PROGRAM F33_OuterPrinters
VAR
	aSquareWave		 		: ARRAY[1..2] OF  FB_SquareWave;
	aOuterCodeGenerator 		: ARRAY[1..2] OF  FB_CODE_OuterCodeGenerator;
	aSelectCommand	 		: ARRAY[1..2] OF  FB_PRINTER_SelectCommand;

	aLabelPrintCtrl				: ARRAY[1..2] OF  RS;
	aLabelApplyCtrl			: ARRAY[1..2] OF  RS;

	tonLoweratorAtConstSpeed	: TON;
	rsInhibitLabbeller1Apply		: RS	;
	rsInhibitLabbeller2Apply		: RS	;

	sAppendedString				: T_LongSTRING;
	
	fbDebugCNT				: FB_DEBUG_CounterArray;
	aCNTDebug				: ARRAY [1..10] OF UDINT;
	bResetCNT				: BOOL;
	bEnableResendCommand		: BOOL;
	rtEncoder	: R_TRIG;
END_VAR
VAR // added by the converter: edge detectors and wires of the graphical bodies
    _w1, _w2, _w3, _w4, _w5, _w6 : BOOL;
END_VAR

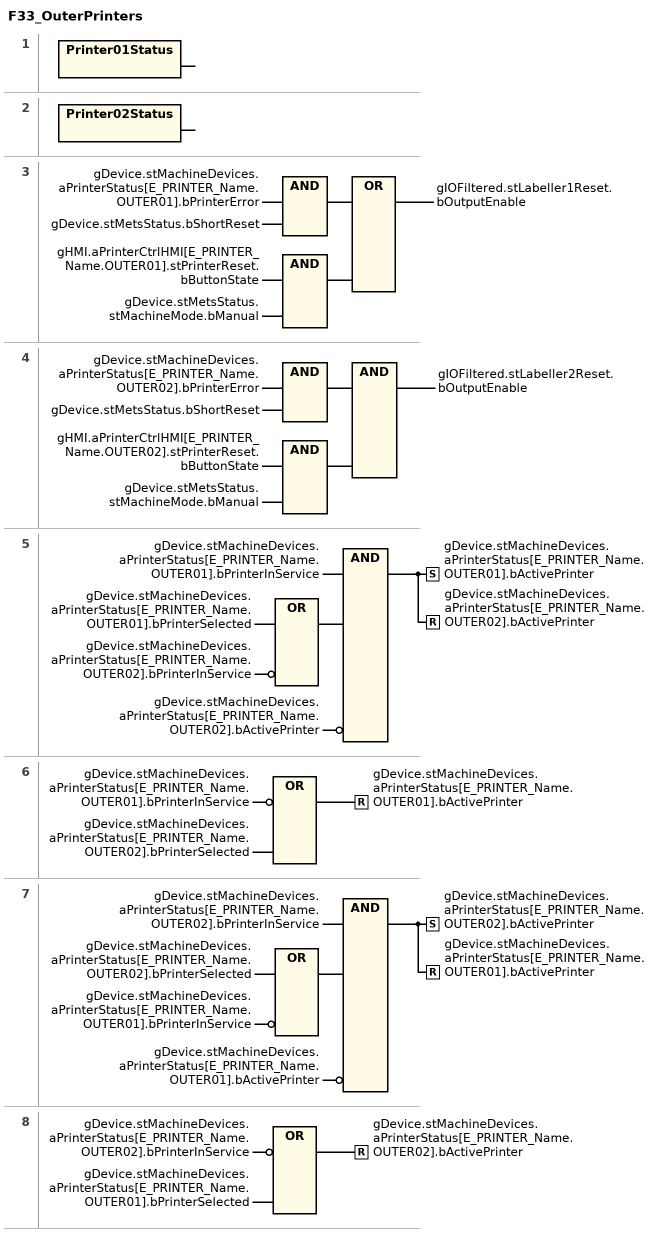
// NETWORK 1
Printer01Status();

// NETWORK 2
Printer02Status();

// NETWORK 3
gIOFiltered.stLabeller1Reset.bOutputEnable := gDevice.stMachineDevices.aPrinterStatus[E_PRINTER_Name.OUTER01].bPrinterError AND gDevice.stMetsStatus.bShortReset OR gHMI.aPrinterCtrlHMI[E_PRINTER_Name.OUTER01].stPrinterReset.bButtonState AND gDevice.stMetsStatus.stMachineMode.bManual;

// NETWORK 4
gIOFiltered.stLabeller2Reset.bOutputEnable := (gDevice.stMachineDevices.aPrinterStatus[E_PRINTER_Name.OUTER02].bPrinterError AND gDevice.stMetsStatus.bShortReset) AND (gHMI.aPrinterCtrlHMI[E_PRINTER_Name.OUTER02].stPrinterReset.bButtonState AND gDevice.stMetsStatus.stMachineMode.bManual);

// NETWORK 5
_w1 := gDevice.stMachineDevices.aPrinterStatus[E_PRINTER_Name.OUTER01].bPrinterInService AND (gDevice.stMachineDevices.aPrinterStatus[E_PRINTER_Name.OUTER01].bPrinterSelected OR NOT gDevice.stMachineDevices.aPrinterStatus[E_PRINTER_Name.OUTER02].bPrinterInService) AND NOT gDevice.stMachineDevices.aPrinterStatus[E_PRINTER_Name.OUTER02].bActivePrinter;
gDevice.stMachineDevices.aPrinterStatus[E_PRINTER_Name.OUTER01].bActivePrinter S= _w1;
gDevice.stMachineDevices.aPrinterStatus[E_PRINTER_Name.OUTER02].bActivePrinter R= _w1;

// NETWORK 6
gDevice.stMachineDevices.aPrinterStatus[E_PRINTER_Name.OUTER01].bActivePrinter R= NOT gDevice.stMachineDevices.aPrinterStatus[E_PRINTER_Name.OUTER01].bPrinterInService OR gDevice.stMachineDevices.aPrinterStatus[E_PRINTER_Name.OUTER02].bPrinterSelected;

// NETWORK 7
_w2 := gDevice.stMachineDevices.aPrinterStatus[E_PRINTER_Name.OUTER02].bPrinterInService AND (gDevice.stMachineDevices.aPrinterStatus[E_PRINTER_Name.OUTER02].bPrinterSelected OR NOT gDevice.stMachineDevices.aPrinterStatus[E_PRINTER_Name.OUTER01].bPrinterInService) AND NOT gDevice.stMachineDevices.aPrinterStatus[E_PRINTER_Name.OUTER01].bActivePrinter;
gDevice.stMachineDevices.aPrinterStatus[E_PRINTER_Name.OUTER02].bActivePrinter S= _w2;
gDevice.stMachineDevices.aPrinterStatus[E_PRINTER_Name.OUTER01].bActivePrinter R= _w2;

// NETWORK 8
gDevice.stMachineDevices.aPrinterStatus[E_PRINTER_Name.OUTER02].bActivePrinter R= NOT gDevice.stMachineDevices.aPrinterStatus[E_PRINTER_Name.OUTER02].bPrinterInService OR gDevice.stMachineDevices.aPrinterStatus[E_PRINTER_Name.OUTER01].bPrinterSelected;

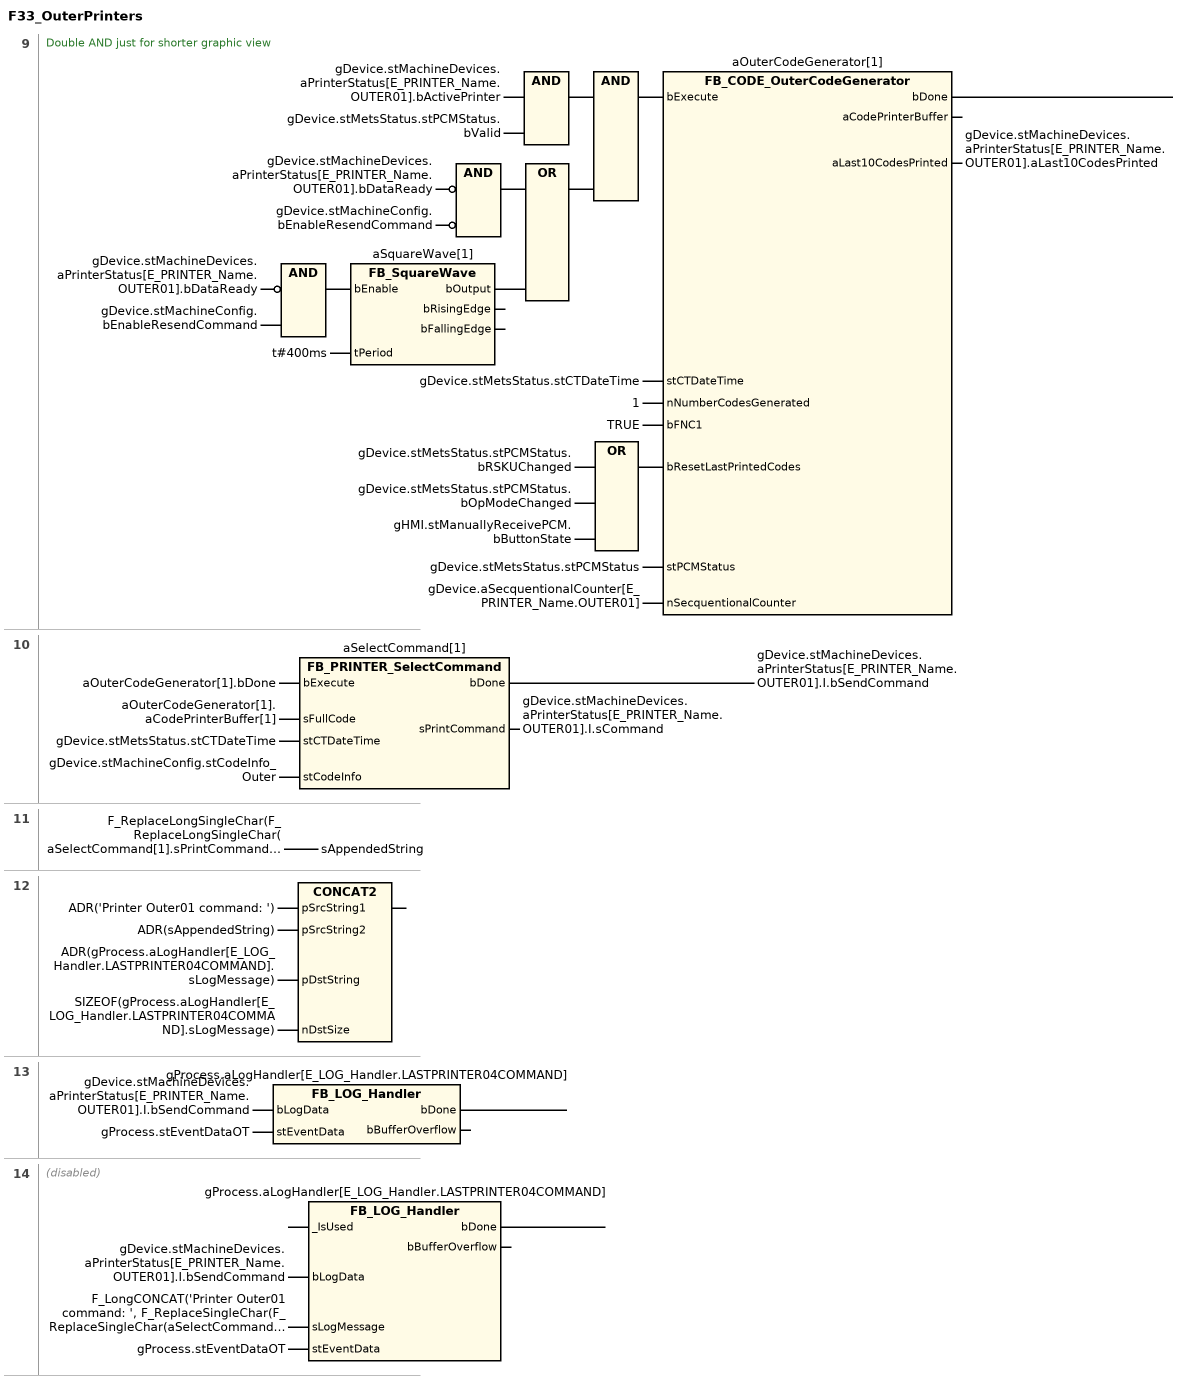
// NETWORK 9
// Double AND just for shorter graphic view
aSquareWave[1](bEnable := NOT gDevice.stMachineDevices.aPrinterStatus[E_PRINTER_Name.OUTER01].bDataReady AND gDevice.stMachineConfig.bEnableResendCommand, tPeriod := t#400ms); // FB_SquareWave
aOuterCodeGenerator[1](
    bExecute := (gDevice.stMachineDevices.aPrinterStatus[E_PRINTER_Name.OUTER01].bActivePrinter AND gDevice.stMetsStatus.stPCMStatus.bValid) AND (NOT gDevice.stMachineDevices.aPrinterStatus[E_PRINTER_Name.OUTER01].bDataReady AND NOT gDevice.stMachineConfig.bEnableResendCommand OR aSquareWave[1].bOutput),
    stCTDateTime := gDevice.stMetsStatus.stCTDateTime,
    nNumberCodesGenerated := 1,
    bFNC1 := TRUE,
    bResetLastPrintedCodes := gDevice.stMetsStatus.stPCMStatus.bRSKUChanged OR gDevice.stMetsStatus.stPCMStatus.bOpModeChanged OR gHMI.stManuallyReceivePCM.bButtonState,
    stPCMStatus := gDevice.stMetsStatus.stPCMStatus,
    nSecquentionalCounter := gDevice.aSecquentionalCounter[E_PRINTER_Name.OUTER01],
    aLast10CodesPrinted => gDevice.stMachineDevices.aPrinterStatus[E_PRINTER_Name.OUTER01].aLast10CodesPrinted); // FB_CODE_OuterCodeGenerator

// NETWORK 10
aSelectCommand[1](
    bExecute := aOuterCodeGenerator[1].bDone,
    sFullCode := aOuterCodeGenerator[1].aCodePrinterBuffer[1],
    stCTDateTime := gDevice.stMetsStatus.stCTDateTime,
    stCodeInfo := gDevice.stMachineConfig.stCodeInfo_Outer,
    sPrintCommand => gDevice.stMachineDevices.aPrinterStatus[E_PRINTER_Name.OUTER01].I.sCommand); // FB_PRINTER_SelectCommand
gDevice.stMachineDevices.aPrinterStatus[E_PRINTER_Name.OUTER01].I.bSendCommand := aSelectCommand[1].bDone;

// NETWORK 11
sAppendedString := F_ReplaceLongSingleChar(F_ReplaceLongSingleChar(aSelectCommand[1].sPrintCommand,'$N','_'),'$R','_');

// NETWORK 12
CONCAT2(pSrcString1 := ADR('Printer Outer01 command: '), pSrcString2 := ADR(sAppendedString), pDstString := ADR(gProcess.aLogHandler[E_LOG_Handler.LASTPRINTER04COMMAND].sLogMessage), nDstSize := SIZEOF(gProcess.aLogHandler[E_LOG_Handler.LASTPRINTER04COMMAND].sLogMessage));

// NETWORK 13
gProcess.aLogHandler[E_LOG_Handler.LASTPRINTER04COMMAND](bLogData := gDevice.stMachineDevices.aPrinterStatus[E_PRINTER_Name.OUTER01].I.bSendCommand, stEventData := gProcess.stEventDataOT); // FB_LOG_Handler

// NETWORK 14 (disabled)
// gProcess.aLogHandler[E_LOG_Handler.LASTPRINTER04COMMAND](
//     bLogData := gDevice.stMachineDevices.aPrinterStatus[E_PRINTER_Name.OUTER01].I.bSendCommand,
//     sLogMessage := F_LongCONCAT('Printer Outer01 command: ', F_ReplaceSingleChar(F_ReplaceSingleChar(aSelectCommand[1].sPrintCommand, '$N', '_' ), '$R', '_')),
//     stEventData := gProcess.stEventDataOT); // FB_LOG_Handler

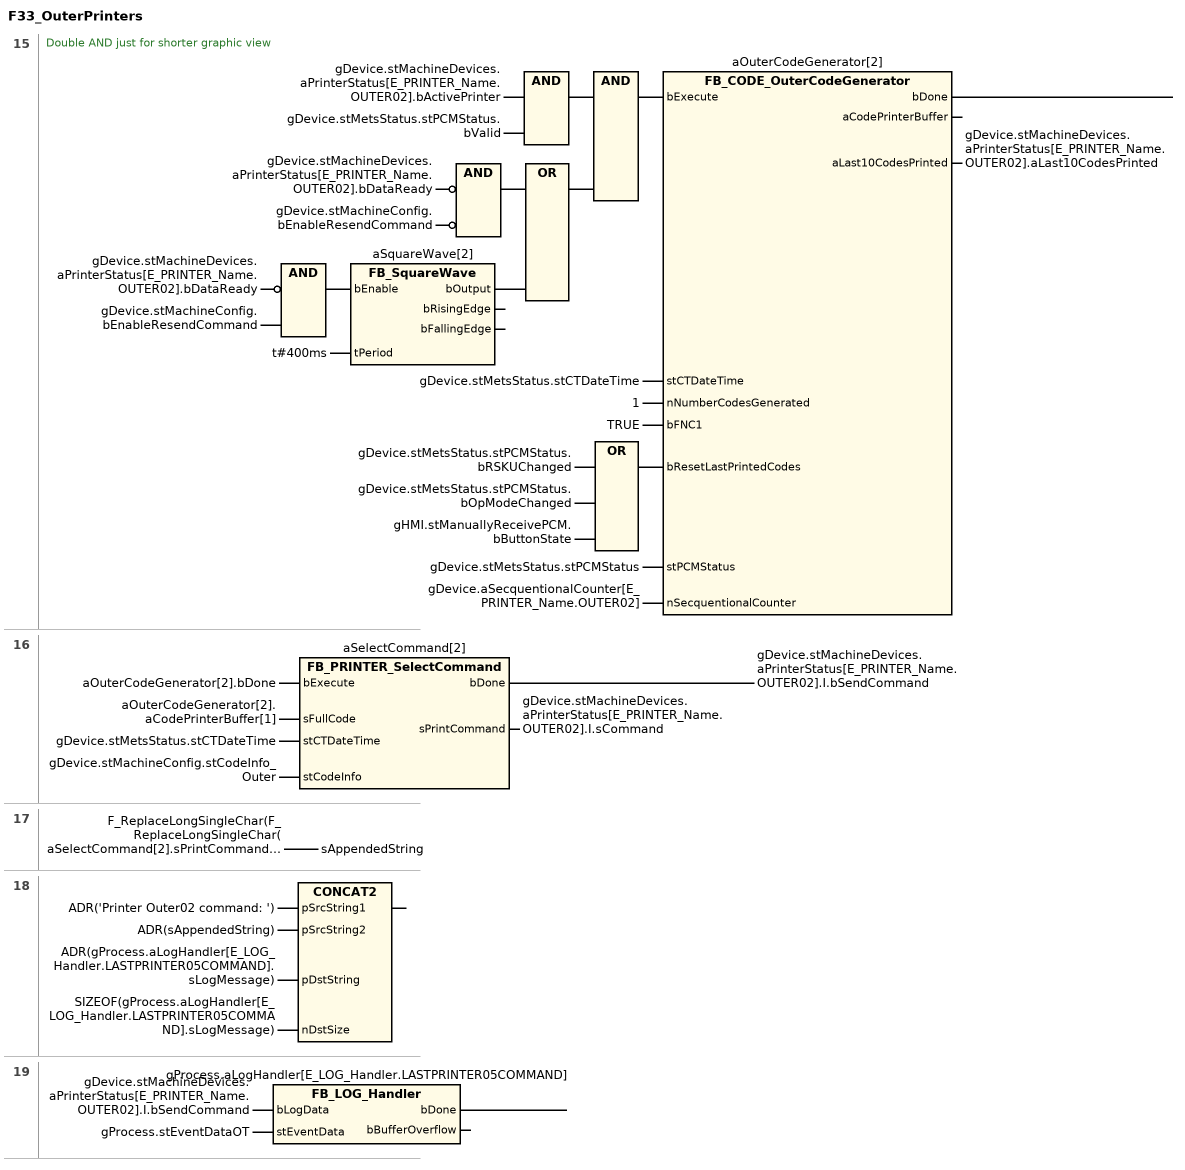
// NETWORK 15
// Double AND just for shorter graphic view
aSquareWave[2](bEnable := NOT gDevice.stMachineDevices.aPrinterStatus[E_PRINTER_Name.OUTER02].bDataReady AND gDevice.stMachineConfig.bEnableResendCommand, tPeriod := t#400ms); // FB_SquareWave
aOuterCodeGenerator[2](
    bExecute := (gDevice.stMachineDevices.aPrinterStatus[E_PRINTER_Name.OUTER02].bActivePrinter AND gDevice.stMetsStatus.stPCMStatus.bValid) AND (NOT gDevice.stMachineDevices.aPrinterStatus[E_PRINTER_Name.OUTER02].bDataReady AND NOT gDevice.stMachineConfig.bEnableResendCommand OR aSquareWave[2].bOutput),
    stCTDateTime := gDevice.stMetsStatus.stCTDateTime,
    nNumberCodesGenerated := 1,
    bFNC1 := TRUE,
    bResetLastPrintedCodes := gDevice.stMetsStatus.stPCMStatus.bRSKUChanged OR gDevice.stMetsStatus.stPCMStatus.bOpModeChanged OR gHMI.stManuallyReceivePCM.bButtonState,
    stPCMStatus := gDevice.stMetsStatus.stPCMStatus,
    nSecquentionalCounter := gDevice.aSecquentionalCounter[E_PRINTER_Name.OUTER02],
    aLast10CodesPrinted => gDevice.stMachineDevices.aPrinterStatus[E_PRINTER_Name.OUTER02].aLast10CodesPrinted); // FB_CODE_OuterCodeGenerator

// NETWORK 16
aSelectCommand[2](
    bExecute := aOuterCodeGenerator[2].bDone,
    sFullCode := aOuterCodeGenerator[2].aCodePrinterBuffer[1],
    stCTDateTime := gDevice.stMetsStatus.stCTDateTime,
    stCodeInfo := gDevice.stMachineConfig.stCodeInfo_Outer,
    sPrintCommand => gDevice.stMachineDevices.aPrinterStatus[E_PRINTER_Name.OUTER02].I.sCommand); // FB_PRINTER_SelectCommand
gDevice.stMachineDevices.aPrinterStatus[E_PRINTER_Name.OUTER02].I.bSendCommand := aSelectCommand[2].bDone;

// NETWORK 17
sAppendedString := F_ReplaceLongSingleChar(F_ReplaceLongSingleChar(aSelectCommand[2].sPrintCommand,'$N','_'),'$R','_');

// NETWORK 18
CONCAT2(pSrcString1 := ADR('Printer Outer02 command: '), pSrcString2 := ADR(sAppendedString), pDstString := ADR(gProcess.aLogHandler[E_LOG_Handler.LASTPRINTER05COMMAND].sLogMessage), nDstSize := SIZEOF(gProcess.aLogHandler[E_LOG_Handler.LASTPRINTER05COMMAND].sLogMessage));

// NETWORK 19
gProcess.aLogHandler[E_LOG_Handler.LASTPRINTER05COMMAND](bLogData := gDevice.stMachineDevices.aPrinterStatus[E_PRINTER_Name.OUTER02].I.bSendCommand, stEventData := gProcess.stEventDataOT); // FB_LOG_Handler

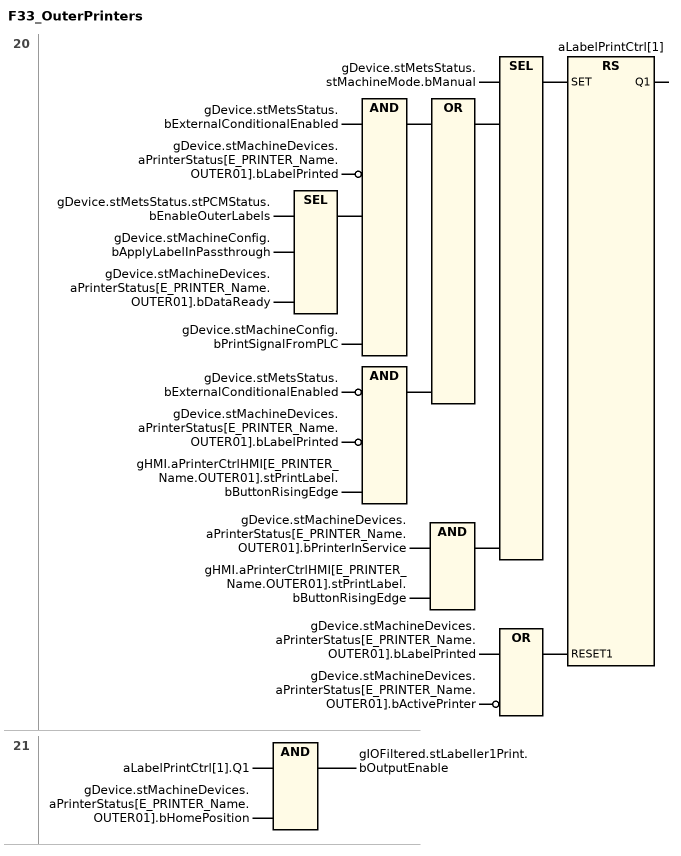
// NETWORK 20
aLabelPrintCtrl[1](SET := SEL(gDevice.stMetsStatus.stMachineMode.bManual, gDevice.stMetsStatus.bExternalConditionalEnabled AND NOT gDevice.stMachineDevices.aPrinterStatus[E_PRINTER_Name.OUTER01].bLabelPrinted AND SEL(gDevice.stMetsStatus.stPCMStatus.bEnableOuterLabels, gDevice.stMachineConfig.bApplyLabelInPassthrough, gDevice.stMachineDevices.aPrinterStatus[E_PRINTER_Name.OUTER01].bDataReady) AND gDevice.stMachineConfig.bPrintSignalFromPLC OR NOT gDevice.stMetsStatus.bExternalConditionalEnabled AND NOT gDevice.stMachineDevices.aPrinterStatus[E_PRINTER_Name.OUTER01].bLabelPrinted AND gHMI.aPrinterCtrlHMI[E_PRINTER_Name.OUTER01].stPrintLabel.bButtonRisingEdge, gDevice.stMachineDevices.aPrinterStatus[E_PRINTER_Name.OUTER01].bPrinterInService AND gHMI.aPrinterCtrlHMI[E_PRINTER_Name.OUTER01].stPrintLabel.bButtonRisingEdge), RESET1 := gDevice.stMachineDevices.aPrinterStatus[E_PRINTER_Name.OUTER01].bLabelPrinted OR NOT gDevice.stMachineDevices.aPrinterStatus[E_PRINTER_Name.OUTER01].bActivePrinter); // RS

// NETWORK 21
gIOFiltered.stLabeller1Print.bOutputEnable := aLabelPrintCtrl[1].Q1 AND gDevice.stMachineDevices.aPrinterStatus[E_PRINTER_Name.OUTER01].bHomePosition;

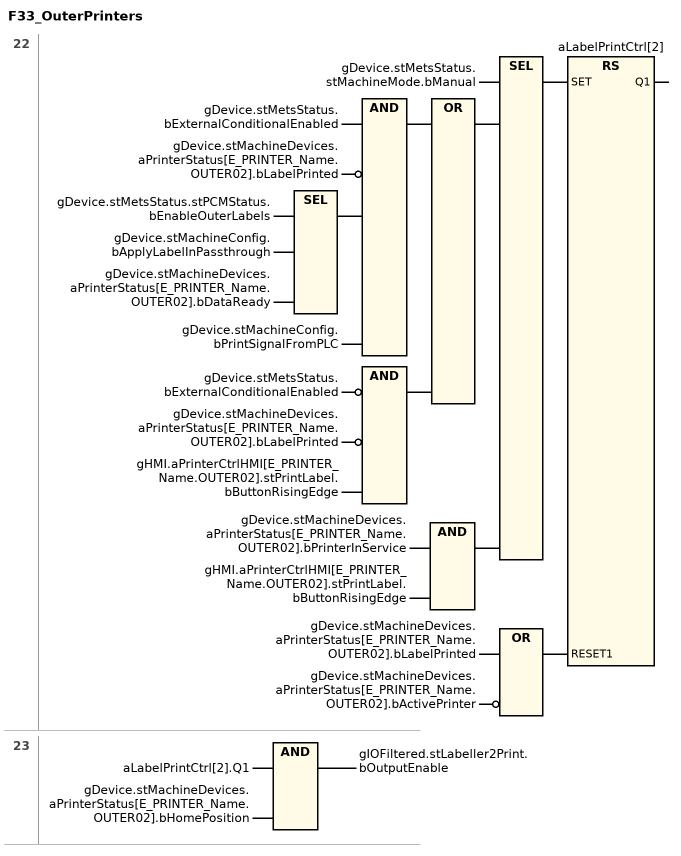
// NETWORK 22
aLabelPrintCtrl[2](SET := SEL(gDevice.stMetsStatus.stMachineMode.bManual, gDevice.stMetsStatus.bExternalConditionalEnabled AND NOT gDevice.stMachineDevices.aPrinterStatus[E_PRINTER_Name.OUTER02].bLabelPrinted AND SEL(gDevice.stMetsStatus.stPCMStatus.bEnableOuterLabels, gDevice.stMachineConfig.bApplyLabelInPassthrough, gDevice.stMachineDevices.aPrinterStatus[E_PRINTER_Name.OUTER02].bDataReady) AND gDevice.stMachineConfig.bPrintSignalFromPLC OR NOT gDevice.stMetsStatus.bExternalConditionalEnabled AND NOT gDevice.stMachineDevices.aPrinterStatus[E_PRINTER_Name.OUTER02].bLabelPrinted AND gHMI.aPrinterCtrlHMI[E_PRINTER_Name.OUTER02].stPrintLabel.bButtonRisingEdge, gDevice.stMachineDevices.aPrinterStatus[E_PRINTER_Name.OUTER02].bPrinterInService AND gHMI.aPrinterCtrlHMI[E_PRINTER_Name.OUTER02].stPrintLabel.bButtonRisingEdge), RESET1 := gDevice.stMachineDevices.aPrinterStatus[E_PRINTER_Name.OUTER02].bLabelPrinted OR NOT gDevice.stMachineDevices.aPrinterStatus[E_PRINTER_Name.OUTER02].bActivePrinter); // RS

// NETWORK 23
gIOFiltered.stLabeller2Print.bOutputEnable := aLabelPrintCtrl[2].Q1 AND gDevice.stMachineDevices.aPrinterStatus[E_PRINTER_Name.OUTER02].bHomePosition;

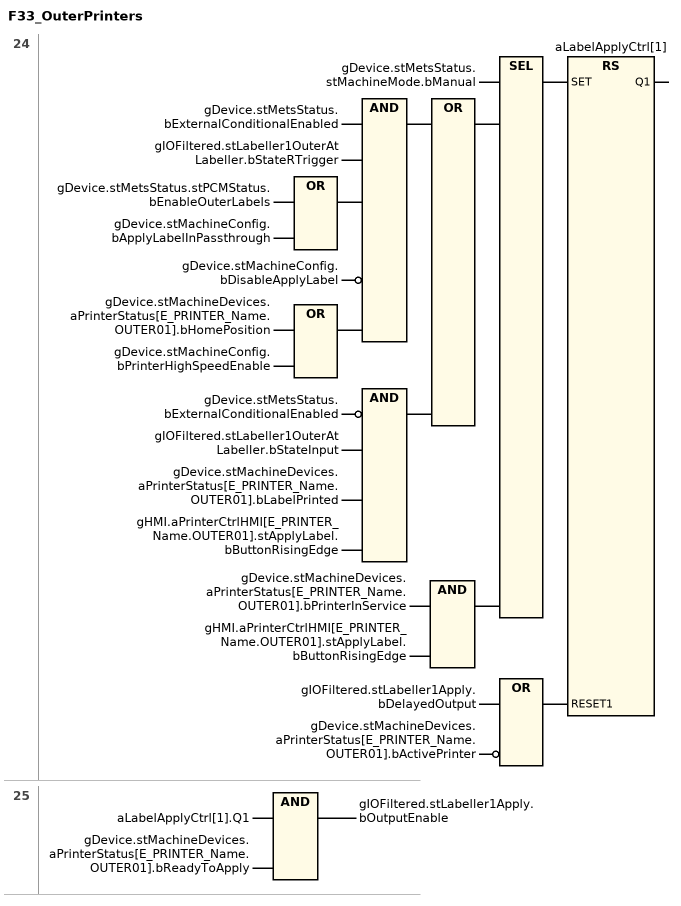
// NETWORK 24
aLabelApplyCtrl[1](SET := SEL(gDevice.stMetsStatus.stMachineMode.bManual, gDevice.stMetsStatus.bExternalConditionalEnabled AND gIOFiltered.stLabeller1OuterAtLabeller.bStateRTrigger AND (gDevice.stMetsStatus.stPCMStatus.bEnableOuterLabels OR gDevice.stMachineConfig.bApplyLabelInPassthrough) AND NOT gDevice.stMachineConfig.bDisableApplyLabel AND (gDevice.stMachineDevices.aPrinterStatus[E_PRINTER_Name.OUTER01].bHomePosition OR gDevice.stMachineConfig.bPrinterHighSpeedEnable) OR NOT gDevice.stMetsStatus.bExternalConditionalEnabled AND gIOFiltered.stLabeller1OuterAtLabeller.bStateInput AND gDevice.stMachineDevices.aPrinterStatus[E_PRINTER_Name.OUTER01].bLabelPrinted AND gHMI.aPrinterCtrlHMI[E_PRINTER_Name.OUTER01].stApplyLabel.bButtonRisingEdge, gDevice.stMachineDevices.aPrinterStatus[E_PRINTER_Name.OUTER01].bPrinterInService AND gHMI.aPrinterCtrlHMI[E_PRINTER_Name.OUTER01].stApplyLabel.bButtonRisingEdge), RESET1 := gIOFiltered.stLabeller1Apply.bDelayedOutput OR NOT gDevice.stMachineDevices.aPrinterStatus[E_PRINTER_Name.OUTER01].bActivePrinter); // RS

// NETWORK 25
gIOFiltered.stLabeller1Apply.bOutputEnable := aLabelApplyCtrl[1].Q1 AND gDevice.stMachineDevices.aPrinterStatus[E_PRINTER_Name.OUTER01].bReadyToApply;

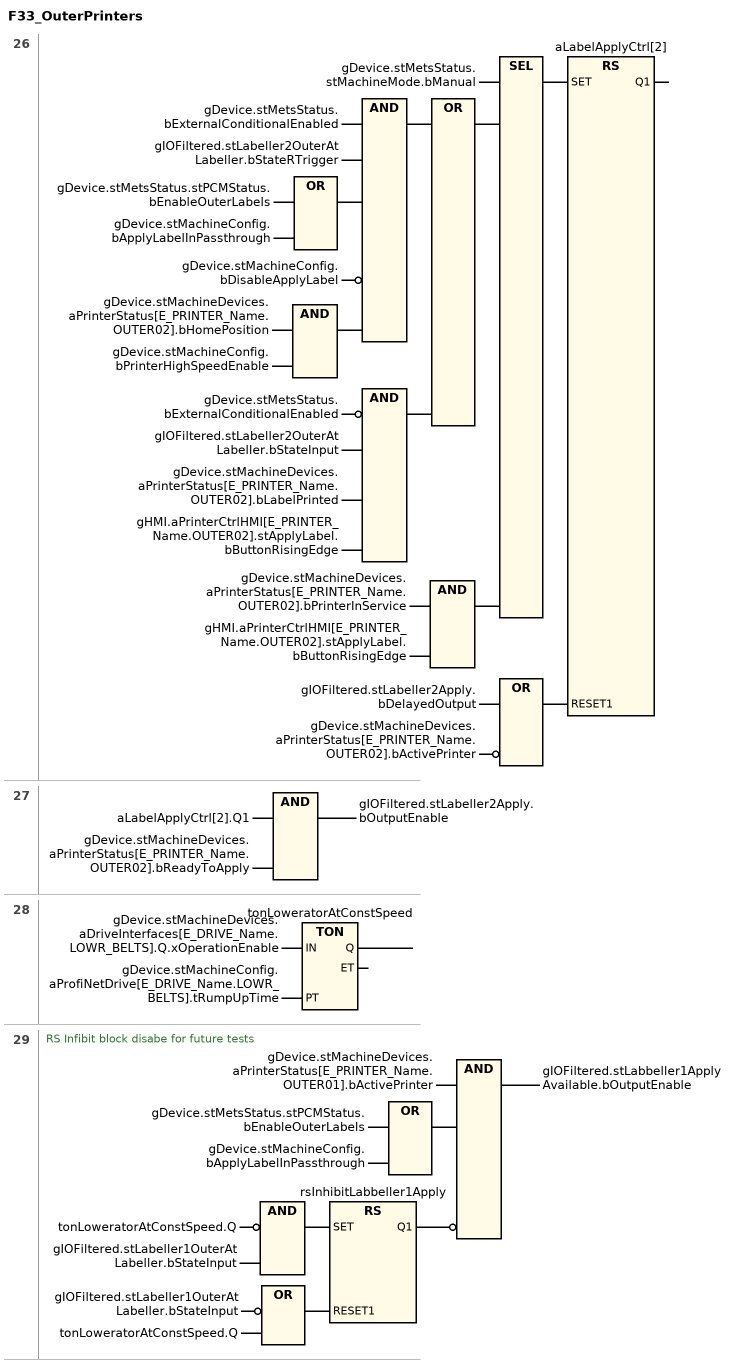
// NETWORK 26
aLabelApplyCtrl[2](SET := SEL(gDevice.stMetsStatus.stMachineMode.bManual, gDevice.stMetsStatus.bExternalConditionalEnabled AND gIOFiltered.stLabeller2OuterAtLabeller.bStateRTrigger AND (gDevice.stMetsStatus.stPCMStatus.bEnableOuterLabels OR gDevice.stMachineConfig.bApplyLabelInPassthrough) AND NOT gDevice.stMachineConfig.bDisableApplyLabel AND (gDevice.stMachineDevices.aPrinterStatus[E_PRINTER_Name.OUTER02].bHomePosition AND gDevice.stMachineConfig.bPrinterHighSpeedEnable) OR NOT gDevice.stMetsStatus.bExternalConditionalEnabled AND gIOFiltered.stLabeller2OuterAtLabeller.bStateInput AND gDevice.stMachineDevices.aPrinterStatus[E_PRINTER_Name.OUTER02].bLabelPrinted AND gHMI.aPrinterCtrlHMI[E_PRINTER_Name.OUTER02].stApplyLabel.bButtonRisingEdge, gDevice.stMachineDevices.aPrinterStatus[E_PRINTER_Name.OUTER02].bPrinterInService AND gHMI.aPrinterCtrlHMI[E_PRINTER_Name.OUTER02].stApplyLabel.bButtonRisingEdge), RESET1 := gIOFiltered.stLabeller2Apply.bDelayedOutput OR NOT gDevice.stMachineDevices.aPrinterStatus[E_PRINTER_Name.OUTER02].bActivePrinter); // RS

// NETWORK 27
gIOFiltered.stLabeller2Apply.bOutputEnable := aLabelApplyCtrl[2].Q1 AND gDevice.stMachineDevices.aPrinterStatus[E_PRINTER_Name.OUTER02].bReadyToApply;

// NETWORK 28
tonLoweratorAtConstSpeed(IN := gDevice.stMachineDevices.aDriveInterfaces[E_DRIVE_Name.LOWR_BELTS].Q.xOperationEnable, PT := gDevice.stMachineConfig.aProfiNetDrive[E_DRIVE_Name.LOWR_BELTS].tRumpUpTime); // TON

// NETWORK 29
// RS Infibit block disabe for future tests
rsInhibitLabbeller1Apply(SET := NOT tonLoweratorAtConstSpeed.Q AND gIOFiltered.stLabeller1OuterAtLabeller.bStateInput, RESET1 := NOT gIOFiltered.stLabeller1OuterAtLabeller.bStateInput OR tonLoweratorAtConstSpeed.Q); // RS
gIOFiltered.stLabbeller1ApplyAvailable.bOutputEnable := gDevice.stMachineDevices.aPrinterStatus[E_PRINTER_Name.OUTER01].bActivePrinter AND (gDevice.stMetsStatus.stPCMStatus.bEnableOuterLabels OR gDevice.stMachineConfig.bApplyLabelInPassthrough) AND NOT rsInhibitLabbeller1Apply.Q1;

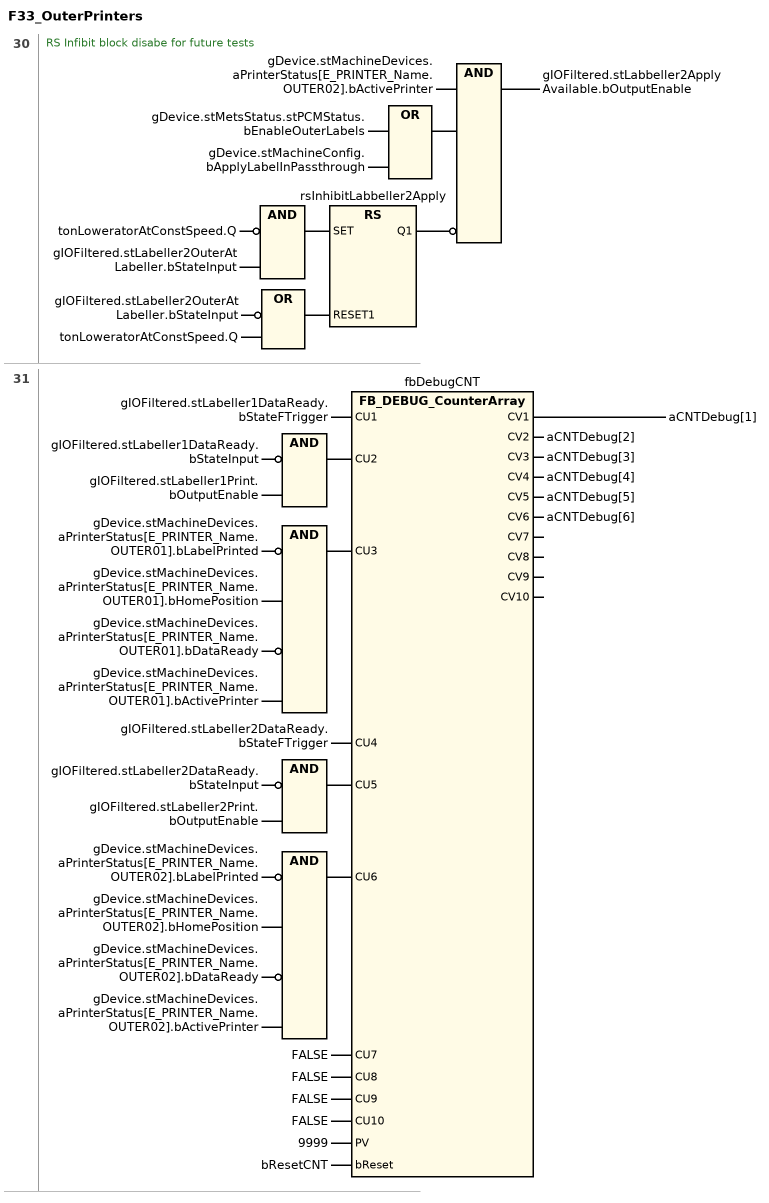
// NETWORK 30
// RS Infibit block disabe for future tests
rsInhibitLabbeller2Apply(SET := NOT tonLoweratorAtConstSpeed.Q AND gIOFiltered.stLabeller2OuterAtLabeller.bStateInput, RESET1 := NOT gIOFiltered.stLabeller2OuterAtLabeller.bStateInput OR tonLoweratorAtConstSpeed.Q); // RS
gIOFiltered.stLabbeller2ApplyAvailable.bOutputEnable := gDevice.stMachineDevices.aPrinterStatus[E_PRINTER_Name.OUTER02].bActivePrinter AND (gDevice.stMetsStatus.stPCMStatus.bEnableOuterLabels OR gDevice.stMachineConfig.bApplyLabelInPassthrough) AND NOT rsInhibitLabbeller2Apply.Q1;

// NETWORK 31
fbDebugCNT(
    CU1 := gIOFiltered.stLabeller1DataReady.bStateFTrigger,
    CU2 := NOT gIOFiltered.stLabeller1DataReady.bStateInput AND gIOFiltered.stLabeller1Print.bOutputEnable,
    CU3 := NOT gDevice.stMachineDevices.aPrinterStatus[E_PRINTER_Name.OUTER01].bLabelPrinted AND gDevice.stMachineDevices.aPrinterStatus[E_PRINTER_Name.OUTER01].bHomePosition AND NOT gDevice.stMachineDevices.aPrinterStatus[E_PRINTER_Name.OUTER01].bDataReady AND gDevice.stMachineDevices.aPrinterStatus[E_PRINTER_Name.OUTER01].bActivePrinter,
    CU4 := gIOFiltered.stLabeller2DataReady.bStateFTrigger,
    CU5 := NOT gIOFiltered.stLabeller2DataReady.bStateInput AND gIOFiltered.stLabeller2Print.bOutputEnable,
    CU6 := NOT gDevice.stMachineDevices.aPrinterStatus[E_PRINTER_Name.OUTER02].bLabelPrinted AND gDevice.stMachineDevices.aPrinterStatus[E_PRINTER_Name.OUTER02].bHomePosition AND NOT gDevice.stMachineDevices.aPrinterStatus[E_PRINTER_Name.OUTER02].bDataReady AND gDevice.stMachineDevices.aPrinterStatus[E_PRINTER_Name.OUTER02].bActivePrinter,
    CU7 := FALSE,
    CU8 := FALSE,
    CU9 := FALSE,
    CU10 := FALSE,
    PV := 9999,
    bReset := bResetCNT,
    CV2 => aCNTDebug[2],
    CV3 => aCNTDebug[3],
    CV4 => aCNTDebug[4],
    CV5 => aCNTDebug[5],
    CV6 => aCNTDebug[6]); // FB_DEBUG_CounterArray
aCNTDebug[1] := fbDebugCNT.CV1;

ACTION Printer01Status:
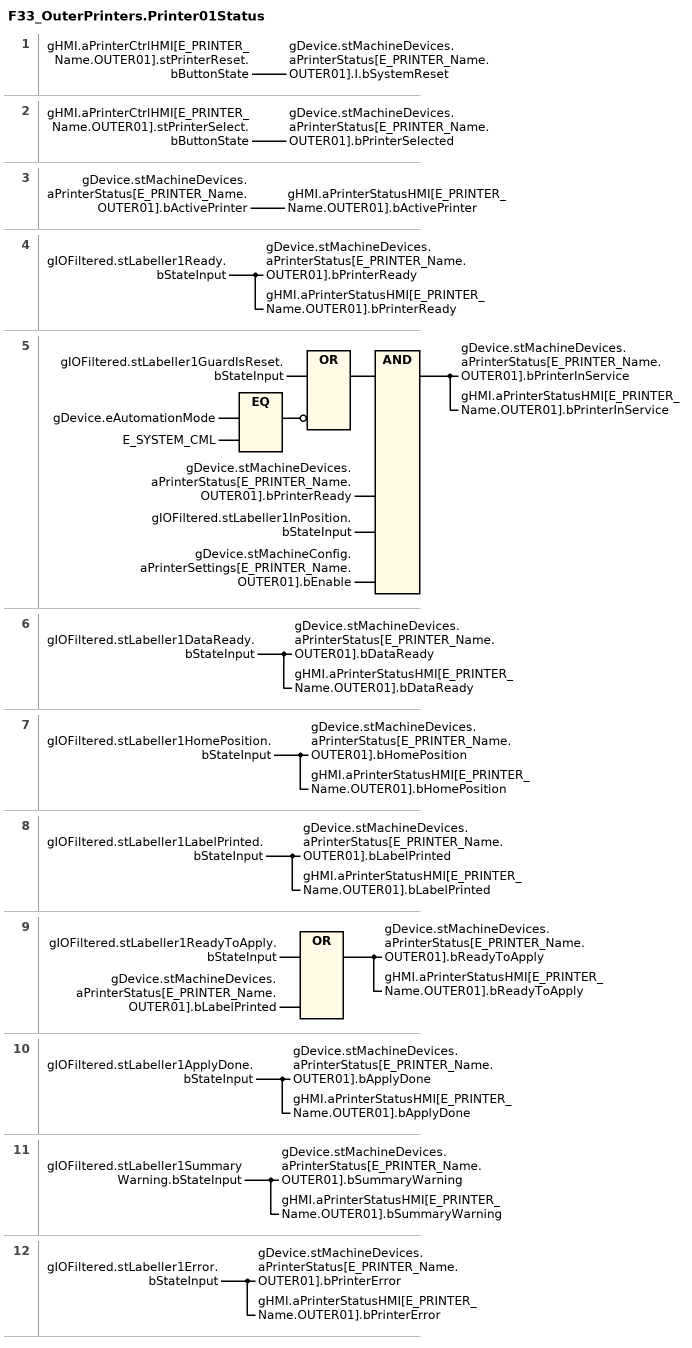
// NETWORK 1
gDevice.stMachineDevices.aPrinterStatus[E_PRINTER_Name.OUTER01].I.bSystemReset := gHMI.aPrinterCtrlHMI[E_PRINTER_Name.OUTER01].stPrinterReset.bButtonState;

// NETWORK 2
gDevice.stMachineDevices.aPrinterStatus[E_PRINTER_Name.OUTER01].bPrinterSelected := gHMI.aPrinterCtrlHMI[E_PRINTER_Name.OUTER01].stPrinterSelect.bButtonState;

// NETWORK 3
gHMI.aPrinterStatusHMI[E_PRINTER_Name.OUTER01].bActivePrinter := gDevice.stMachineDevices.aPrinterStatus[E_PRINTER_Name.OUTER01].bActivePrinter;

// NETWORK 4
gDevice.stMachineDevices.aPrinterStatus[E_PRINTER_Name.OUTER01].bPrinterReady := gIOFiltered.stLabeller1Ready.bStateInput;
gHMI.aPrinterStatusHMI[E_PRINTER_Name.OUTER01].bPrinterReady := gIOFiltered.stLabeller1Ready.bStateInput;

// NETWORK 5
_w3 := (gIOFiltered.stLabeller1GuardIsReset.bStateInput OR NOT (gDevice.eAutomationMode = E_SYSTEM_CML)) AND gDevice.stMachineDevices.aPrinterStatus[E_PRINTER_Name.OUTER01].bPrinterReady AND gIOFiltered.stLabeller1InPosition.bStateInput AND gDevice.stMachineConfig.aPrinterSettings[E_PRINTER_Name.OUTER01].bEnable;
gDevice.stMachineDevices.aPrinterStatus[E_PRINTER_Name.OUTER01].bPrinterInService := _w3;
gHMI.aPrinterStatusHMI[E_PRINTER_Name.OUTER01].bPrinterInService := _w3;

// NETWORK 6
gDevice.stMachineDevices.aPrinterStatus[E_PRINTER_Name.OUTER01].bDataReady := gIOFiltered.stLabeller1DataReady.bStateInput;
gHMI.aPrinterStatusHMI[E_PRINTER_Name.OUTER01].bDataReady := gIOFiltered.stLabeller1DataReady.bStateInput;

// NETWORK 7
gDevice.stMachineDevices.aPrinterStatus[E_PRINTER_Name.OUTER01].bHomePosition := gIOFiltered.stLabeller1HomePosition.bStateInput;
gHMI.aPrinterStatusHMI[E_PRINTER_Name.OUTER01].bHomePosition := gIOFiltered.stLabeller1HomePosition.bStateInput;

// NETWORK 8
gDevice.stMachineDevices.aPrinterStatus[E_PRINTER_Name.OUTER01].bLabelPrinted := gIOFiltered.stLabeller1LabelPrinted.bStateInput;
gHMI.aPrinterStatusHMI[E_PRINTER_Name.OUTER01].bLabelPrinted := gIOFiltered.stLabeller1LabelPrinted.bStateInput;

// NETWORK 9
_w4 := gIOFiltered.stLabeller1ReadyToApply.bStateInput OR gDevice.stMachineDevices.aPrinterStatus[E_PRINTER_Name.OUTER01].bLabelPrinted;
gDevice.stMachineDevices.aPrinterStatus[E_PRINTER_Name.OUTER01].bReadyToApply := _w4;
gHMI.aPrinterStatusHMI[E_PRINTER_Name.OUTER01].bReadyToApply := _w4;

// NETWORK 10
gDevice.stMachineDevices.aPrinterStatus[E_PRINTER_Name.OUTER01].bApplyDone := gIOFiltered.stLabeller1ApplyDone.bStateInput;
gHMI.aPrinterStatusHMI[E_PRINTER_Name.OUTER01].bApplyDone := gIOFiltered.stLabeller1ApplyDone.bStateInput;

// NETWORK 11
gDevice.stMachineDevices.aPrinterStatus[E_PRINTER_Name.OUTER01].bSummaryWarning := gIOFiltered.stLabeller1SummaryWarning.bStateInput;
gHMI.aPrinterStatusHMI[E_PRINTER_Name.OUTER01].bSummaryWarning := gIOFiltered.stLabeller1SummaryWarning.bStateInput;

// NETWORK 12
gDevice.stMachineDevices.aPrinterStatus[E_PRINTER_Name.OUTER01].bPrinterError := gIOFiltered.stLabeller1Error.bStateInput;
gHMI.aPrinterStatusHMI[E_PRINTER_Name.OUTER01].bPrinterError := gIOFiltered.stLabeller1Error.bStateInput;
END_ACTION

ACTION Printer02Status:
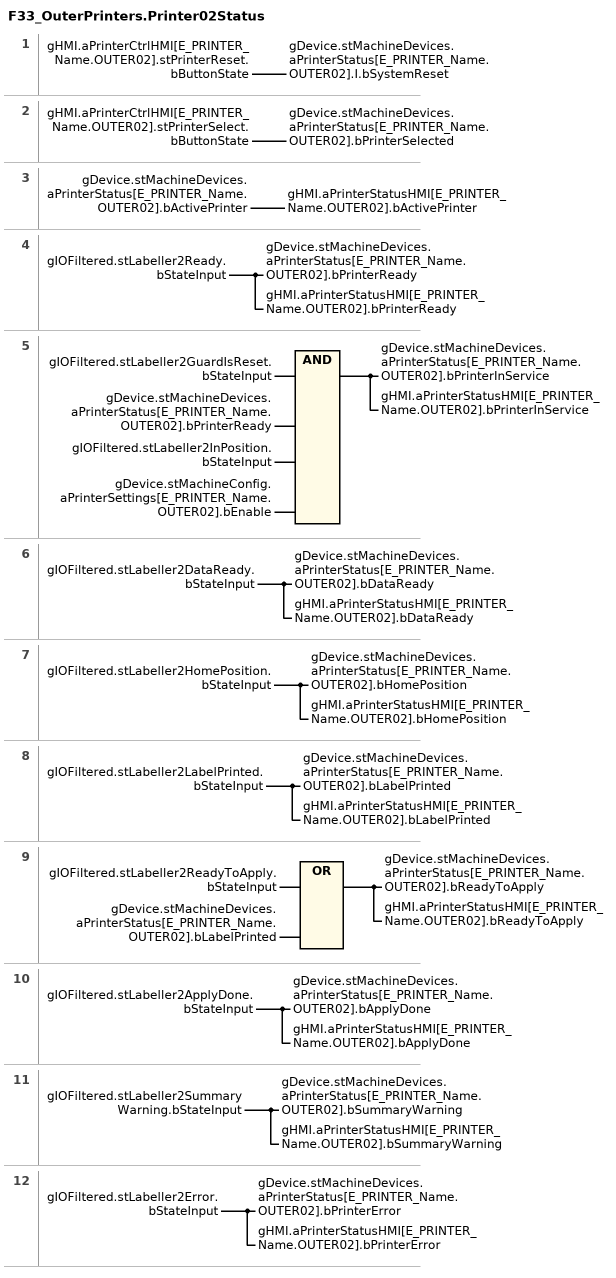
// NETWORK 1
gDevice.stMachineDevices.aPrinterStatus[E_PRINTER_Name.OUTER02].I.bSystemReset := gHMI.aPrinterCtrlHMI[E_PRINTER_Name.OUTER02].stPrinterReset.bButtonState;

// NETWORK 2
gDevice.stMachineDevices.aPrinterStatus[E_PRINTER_Name.OUTER02].bPrinterSelected := gHMI.aPrinterCtrlHMI[E_PRINTER_Name.OUTER02].stPrinterSelect.bButtonState;

// NETWORK 3
gHMI.aPrinterStatusHMI[E_PRINTER_Name.OUTER02].bActivePrinter := gDevice.stMachineDevices.aPrinterStatus[E_PRINTER_Name.OUTER02].bActivePrinter;

// NETWORK 4
gDevice.stMachineDevices.aPrinterStatus[E_PRINTER_Name.OUTER02].bPrinterReady := gIOFiltered.stLabeller2Ready.bStateInput;
gHMI.aPrinterStatusHMI[E_PRINTER_Name.OUTER02].bPrinterReady := gIOFiltered.stLabeller2Ready.bStateInput;

// NETWORK 5
_w5 := gIOFiltered.stLabeller2GuardIsReset.bStateInput AND gDevice.stMachineDevices.aPrinterStatus[E_PRINTER_Name.OUTER02].bPrinterReady AND gIOFiltered.stLabeller2InPosition.bStateInput AND gDevice.stMachineConfig.aPrinterSettings[E_PRINTER_Name.OUTER02].bEnable;
gDevice.stMachineDevices.aPrinterStatus[E_PRINTER_Name.OUTER02].bPrinterInService := _w5;
gHMI.aPrinterStatusHMI[E_PRINTER_Name.OUTER02].bPrinterInService := _w5;

// NETWORK 6
gDevice.stMachineDevices.aPrinterStatus[E_PRINTER_Name.OUTER02].bDataReady := gIOFiltered.stLabeller2DataReady.bStateInput;
gHMI.aPrinterStatusHMI[E_PRINTER_Name.OUTER02].bDataReady := gIOFiltered.stLabeller2DataReady.bStateInput;

// NETWORK 7
gDevice.stMachineDevices.aPrinterStatus[E_PRINTER_Name.OUTER02].bHomePosition := gIOFiltered.stLabeller2HomePosition.bStateInput;
gHMI.aPrinterStatusHMI[E_PRINTER_Name.OUTER02].bHomePosition := gIOFiltered.stLabeller2HomePosition.bStateInput;

// NETWORK 8
gDevice.stMachineDevices.aPrinterStatus[E_PRINTER_Name.OUTER02].bLabelPrinted := gIOFiltered.stLabeller2LabelPrinted.bStateInput;
gHMI.aPrinterStatusHMI[E_PRINTER_Name.OUTER02].bLabelPrinted := gIOFiltered.stLabeller2LabelPrinted.bStateInput;

// NETWORK 9
_w6 := gIOFiltered.stLabeller2ReadyToApply.bStateInput OR gDevice.stMachineDevices.aPrinterStatus[E_PRINTER_Name.OUTER02].bLabelPrinted;
gDevice.stMachineDevices.aPrinterStatus[E_PRINTER_Name.OUTER02].bReadyToApply := _w6;
gHMI.aPrinterStatusHMI[E_PRINTER_Name.OUTER02].bReadyToApply := _w6;

// NETWORK 10
gDevice.stMachineDevices.aPrinterStatus[E_PRINTER_Name.OUTER02].bApplyDone := gIOFiltered.stLabeller2ApplyDone.bStateInput;
gHMI.aPrinterStatusHMI[E_PRINTER_Name.OUTER02].bApplyDone := gIOFiltered.stLabeller2ApplyDone.bStateInput;

// NETWORK 11
gDevice.stMachineDevices.aPrinterStatus[E_PRINTER_Name.OUTER02].bSummaryWarning := gIOFiltered.stLabeller2SummaryWarning.bStateInput;
gHMI.aPrinterStatusHMI[E_PRINTER_Name.OUTER02].bSummaryWarning := gIOFiltered.stLabeller2SummaryWarning.bStateInput;

// NETWORK 12
gDevice.stMachineDevices.aPrinterStatus[E_PRINTER_Name.OUTER02].bPrinterError := gIOFiltered.stLabeller2Error.bStateInput;
gHMI.aPrinterStatusHMI[E_PRINTER_Name.OUTER02].bPrinterError := gIOFiltered.stLabeller2Error.bStateInput;
END_ACTION

END_PROGRAM

(* stored: Version 1.1.0.1
   POU F33_OuterPrinters: Id {c96ed4dd-ce35-4358-9b02-7df8a87f17a3}, SpecialFunc None
   Action Printer01Status: Id {104ab887-f2df-401d-8bd9-7a8dc625d1ee}
   Action Printer02Status: Id {40c3685f-403e-4325-8a8b-f19531f77c14} *)
